{attribute addProperty BoxType "EJ6224-0000-0016"}
{attribute addProperty Id "State_Ch1AT %I*USINT811State_Ch2AT %I*USINT812State_Ch3AT %I*USINT813State_Ch4AT %I*USINT814"}
{attribute addProperty CRC "3183918787"}
{attribute addProperty SizeInBites "32"}
{attribute addProperty SizeInBytes "4"}
TYPE DeviceState_Inputs_BDC6BEC3 :
STRUCT
	{attribute addProperty Name "State_Ch1"}
	State_Ch1 AT %I* : USINT;
	{attribute addProperty Name "State_Ch2"}
	State_Ch2 AT %I* : USINT;
	{attribute addProperty Name "State_Ch3"}
	State_Ch3 AT %I* : USINT;
	{attribute addProperty Name "State_Ch4"}
	State_Ch4 AT %I* : USINT;
END_STRUCT
END_TYPE

(* stored: Version 1.2.0.0, ProductVersion 3.1.4024.9
   DUT DeviceState_Inputs_BDC6BEC3: Id {fc8a8476-72a9-4a36-919e-6304fed3e52a} *)
